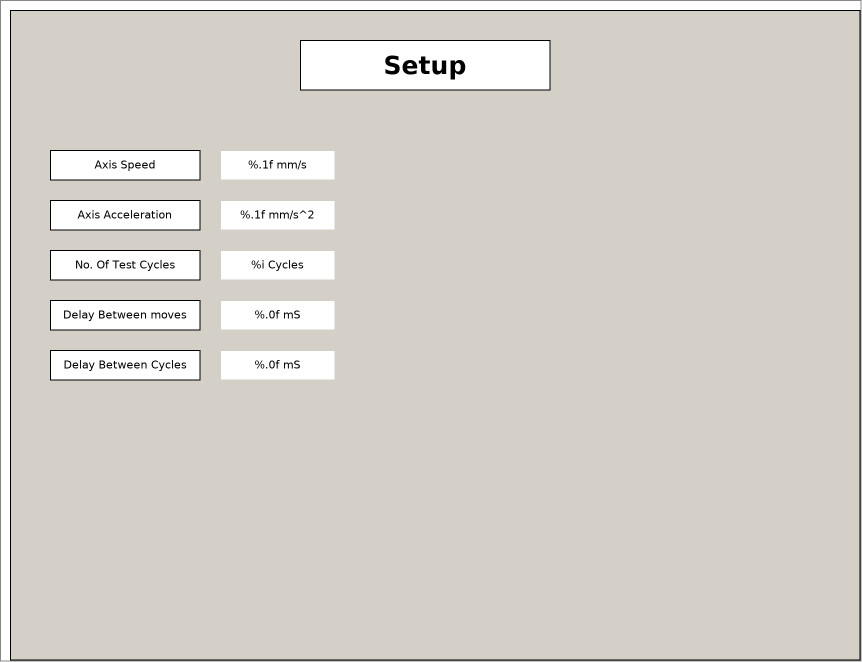
VISUALIZATION Set_Up  // 862x662
    RoundedRectangle (10,10 850x650)
    RoundedRectangle (300,40 250x50), "Setup"
    Rectangle (50,150 150x30), "Axis Speed"
    Textfield (220,150 115x30), "%.1f mm/s", text variable: MAIN.fAxisVelocity
        OnMouseClick: write the text variable via VisuDialogs.Numpad, min 0, max 20, format 1
    Rectangle (50,200 150x30), "Axis Acceleration"
    Textfield (220,200 115x30), "%.1f mm/s^2", text variable: MAIN.fAxisAcceleration
        OnMouseClick: write the text variable via VisuDialogs.Numpad, min 0, max 20, format 1
    Rectangle (50,350 150x30), "Delay Between Cycles"
    Rectangle (50,300 150x30), "Delay Between moves"
    Rectangle (50,250 150x30), "No. Of Test Cycles"
    Textfield (220,350 115x30), "%.0f mS", text variable: MAIN.uInputCycleTime
        OnMouseClick: write the text variable via VisuDialogs.Numpad
    Textfield (220,300 115x30), "%.0f mS", text variable: MAIN.uInputReurnTime
        OnMouseClick: write the text variable via VisuDialogs.Numpad
    Textfield (220,250 115x30), "%i Cycles", text variable: MAIN.iCycleCount
        OnMouseClick: write the text variable via VisuDialogs.Numpad, min 1, max 32000
END_VISUALIZATION

(* stored: Version 1.1.0.1, ProductVersion 3.1.4024.0
   Visu Set_Up: Id {9b47bdc7-a0dd-406d-b2f3-1cff23275595} *)
